(* IEC 61131-3 sources: POMIRTS_lab3/AS/Library/AsHost, 3 files *)

(* ---- AsHost.typ ---- *)
(********************************************************************
 * COPYRIGHT -- Bernecker + Rainer
 ********************************************************************
 * Library: AsHost
 * File: AsHost.typ
 * Author: B+R
 ********************************************************************
 * Data types of library AsHost
 ********************************************************************)

TYPE
	ASHOST_LOCAL_OBJ : STRUCT			(*internal use*)
		StateMan		: UINT;
		ErrMan			: UINT;
		Init			: UDINT;
		END_STRUCT;
END_TYPE

(* ---- AsHost.fun ---- *)
(********************************************************************
 * COPYRIGHT -- Bernecker + Rainer
 ********************************************************************
 * Library: AsHost
 * File: AsHost.fun
 * Author: B+R
 ********************************************************************
 * Functions and function blocks of library AsHost
 ********************************************************************)

FUNCTION_BLOCK HostByName					(*returns the accompanying IP address for the specified host name*)
	VAR_INPUT
		enable       : BOOL;				(*enables execution*)
		pName		 : UDINT;				(*pointer to the name to be resolved, e.g. "sun.galaxy.one"*)
	END_VAR

	VAR
		Obj			 : ASHOST_LOCAL_OBJ;	(*internal variable*)
	END_VAR

	VAR_OUTPUT
		status		 : UINT;				(*execution status: ERR_OK, ERR_FUB_ENABLE_FALSE, 0xXXXX = see help*)
		address		 : UDINT;				(*IP address in HEX format, e.g. "10.43.75.1" -> 0x014B2B0A*)
	END_VAR
END_FUNCTION_BLOCK

FUNCTION_BLOCK HostByAddress				(*returns the accompanying host name for the specified IP address*)
	VAR_INPUT
		enable       : BOOL; 				(*enables execution*)
		address	 	 : UDINT;				(*IP address to be resolved in HEX format, e.g. "10.43.75.1" -> 0x014B2B0A*)
		pName		 : UDINT;				(*pointer to the name buffer*)
		buflng		 : UDINT;				(*length of the buffer*)
	END_VAR

	VAR
		Obj			 : ASHOST_LOCAL_OBJ;	(*internal variable*)
	END_VAR

	VAR_OUTPUT
		status		 : UINT; 				(*execution status: ERR_OK, ERR_FUB_ENABLE_FALSE, 0xXXXX = see help*)
	END_VAR
END_FUNCTION_BLOCK

(* ---- AsHost.var ---- *)
(********************************************************************
 * COPYRIGHT -- Bernecker + Rainer
 ********************************************************************
 * Library: AsHost
 * File: AsHost.var
 * Author: B+R
 ********************************************************************
 * Local variables of library AsHost
 ********************************************************************)

VAR CONSTANT
	ERR_ASHOST_MANAGER		: UINT := 29750;		(*internal manager error*)
	ERR_ASHOST_PARAM_ADDR	: UINT := 29751;		(*specified "address" parameter invalid*)
	ERR_ASHOST_PARAM_BUFLNG : UINT := 29752;		(*specified buffer length too small*)
	ERR_ASHOST_PARAM_NAME	: UINT := 29753;		(*specified "pName" parameter invalid*)
	ERR_ASHOST_RESOLV_ADDR	: UINT := 29754;		(*IP address could not be resolved*)
	ERR_ASHOST_RESOLV_NAME	: UINT := 29755;		(*name could not be resolved*)
END_VAR
